TYPE Debug_ComponentCalls:
STRUCT
	
	//Stn 051 Programs
	CallStn051_20_ReturnBreakStopsGrn: BOOL;
	CallStn051_21_ReturnBreakStopsRed: BOOL;
	
	//Stn 052 Programs
	CallStn052_20_ReceivingBreakStopsGrn: BOOL;
	CallStn052_21_ReceivingBreakStopsRed: BOOL;
	CallStn052_35_Stn123Divert: BOOL;
	CallStn052_36_Stn123MainMergePrestop: BOOL;
	CallStn052_37_Stn123Merge: BOOL;
	CallStn052_40_Stn124Divert: BOOL;
	CallStn052_41_Stn124MainMergePrestop: BOOL;
	CallStn052_42_Stn124Merge: BOOL;
	CallStn052_45_Stn125Divert: BOOL;
	CallStn052_46_Stn125MainMergePrestop: BOOL;
	CallStn052_47_Stn125Merge: BOOL;
	CallStn052_50_Stn126Divert: BOOL;
	CallStn052_51_Stn126MainMergePrestop: BOOL;
	CallStn052_52_Stn126Merge: BOOL;
	
	//Stn 053 Call Programs
	CallStn053_22_EvalBreakStopsBlu: BOOL;
	CallStn053_25_EmptyPuckStorageBreakStop1Red: BOOL;
	CallStn053_26_EmptyPuckStorageBreakStop2Red: BOOL;
	CallStn053_41_BufferRecircMainMergePrestopRed: BOOL;
	CallStn053_42_BufferRecircSpurMergePrestopRed: BOOL;
	CallStn053_43_BufferRecircMergeRed: BOOL;
	CallStn053_45_CleaningRecircExitDivertRed: BOOL;
	CallStn053_97_RedGrnRecircMergePrestopRed: BOOL;
	CallStn053_98_ReceivingBypassExitMergeMainPrestopBlu: BOOL;
	CallStn053_99_ReceivingBypassExitMergeBlu: BOOL;

	//Stn 054 Call Programs
	CallStn054_15_RedGrnRecircMainMergePrestopGrn: BOOL;
	CallStn054_16_RedGrnRecircMerge: BOOL;
	CallStn054_17_RedGrnRecircSpurMergePrestopRed: BOOL;
	CallStn054_22_EvalBreakStopsGrn: BOOL;
	CallStn054_24_EmptyPuckStorageDivertGrn: BOOL;
	CallStn054_25_EmptyPuckStorageBreakStop1Grn: BOOL;
	CallStn054_26_EmptyPuckStorageBreakStop2Grn: BOOL;
	CallStn054_27_EmptyPuckStorageMainMergePrestopGrn: BOOL;
	CallStn054_28_EmptyPuckStorageSpurMergePrestopGrn: BOOL;
	CallStn054_29_EmptyPuckStorageMergeGrn: BOOL;
	CallStn054_30_Stn311Divert: BOOL;
	CallStn054_31_Stn311MergePrestop: BOOL;
	CallStn054_32_Stn311Merge: BOOL;
	CallStn054_40_BufferRecircEntryDivertGrn: BOOL;
	CallStn054_41_BufferRecircMainMergePrestopGrn: BOOL;
	CallStn054_42_BufferRecircSpurMergePrestopGrn: BOOL;
	CallStn054_43_BufferRecircMergeGrn: BOOL;
	CallStn054_45_CleaningRecircExitDivertGrn: BOOL;
	CallStn054_46_CleaningRecircExitMainMergePrestopGrn: BOOL;
	CallStn054_47_CleaningRecircExitSpurMergePrestopGrn: BOOL;
	CallStn054_48_CleaningRecircExitMergeGrn: BOOL;
	CallStn054_50_Stn321Divert: BOOL;
	CallStn054_51_Stn321MainMergePrestop: BOOL;
	CallStn054_52_Stn321Merge: BOOL;
	CallStn054_55_Stn322Divert: BOOL;
	CallStn054_56_Stn322MainMergePrestop: BOOL;
	CallStn054_57_Stn322Merge: BOOL;
	CallStn054_60_Stn331Divert: BOOL;
	CallStn054_61_Stn331MainMergePrestop: BOOL;
	CallStn054_62_Stn331Merge: BOOL;
	CallStn054_65_Stn332Divert: BOOL;
	CallStn054_66_Stn332MainMergePrestop: BOOL;
	CallStn054_67_Stn332Merge: BOOL;
	CallStn054_75_GradingRecircEntryDivertGrn: BOOL;
	CallStn054_76_TestRecircExitMainMergePrestopGrn: BOOL;
	CallStn054_77_TestRecircExitSpurMergePrestopGrn: BOOL;
	CallStn054_78_TestRecircExitMergeGrn: BOOL;
	CallStn054_80_Stn341Divert: BOOL;
	CallStn054_81_Stn341MainMergePrestop: BOOL;
	CallStn054_82_Stn341Merge: BOOL;
	CallStn054_88_Stn351Divert: BOOL;
	CallStn054_89_Stn351MainMergePrestop: BOOL;
	CallStn054_90_Stn351Merge: BOOL;
	CallStn054_91_Stn352Divert: BOOL;
	CallStn054_92_Stn352MainMergePrestop: BOOL;
	CallStn054_93_Stn352Merge: BOOL;
	CallStn054_95_TestRecircEntryDivertGrn: BOOL;
	CallStn054_96_EvalRecircBreakStopsGrn: BOOL;
	
	
	//Stn 055 Red Line Components
	CallStn055_21_StorageBreakStopsRed: BOOL;
	CallStn055_40_StorageBypassDivertRed: BOOL;
	CallStn055_41_StorageBypassMainMergePrestopRed: BOOL;
	CallStn055_42_StorageBypassSpurMergePrestopRed: BOOL;
	CallStn055_43_StorageBypassMergeRed: BOOL;
	CallStn055_45_Stn511Divert: BOOL;
	CallStn055_46_Stn511MainMergePrestop: BOOL;
	CallStn055_47_Stn511Merge: BOOL;
	CallStn055_50_Stn512Divert: BOOL;
	CallStn055_51_Stn512MainMergePrestop: BOOL;
	CallStn055_52_Stn512Merge: BOOL;
		
	//Stn 055 Green Line Components
	CallStn055_20_StorageBreakStopsGrn: BOOL;
	CallStn055_25_StorageBypassDivertGrn: BOOL;
	CallStn055_26_StorageBypassMainMergePrestopGrn: BOOL;
	CallStn055_27_StorageBypassSpurMergePrestopGrn: BOOL;
	CallStn055_28_StorageBypassMergeGrn: BOOL;
	CallStn055_30_Stn411Divert: BOOL;
	CallStn055_31_Stn411MainMergePrestop: BOOL;
	CallStn055_32_Stn411Merge: BOOL;	

END_STRUCT
END_TYPE

(* stored: Version 1.1.0.1, ProductVersion 3.1.4024.6
   DUT Debug_ComponentCalls: Id {17aa2fd4-68ab-4825-8763-c855c1e0aae6} *)
